// TIA Portal project "Omogenizator Miere V18" (V18)

(* hardware
DEVICE "S7-1200 station_1"  S7-1200 Station
   slot 0: "Rack_0"  S7-1200 Rack  Rack  V1.0
   slot 1: "PLC_1"  CPU 1215C DC/DC/Rly  6ES7 215-1HG40-0XB0  V4.6
DEVICE "HMI_1"  TP700 Comfort
   slot 0: "HMI_1"  TP700 Comfort  6AV2 124-0GC01-0AX0  17.0.0.0
   slot 1: "HMI_RT_1"  TP700 Comfort  6AV2 124-0GC01-0AX0  17.0.0.0
   slot 5: "HMI_1.IE_CP_1"  PROFINET Interface  17.0.0.0
      slot 1: "PROFINET Interface_1"  PROFINET Interface
         slot 1: "Port_1"  Port
         slot 2: "Port_2"  Port
   slot 7: "HMI_1.MPI/DP_CP_1"  MPI/DP Interface  17.0.0.0
DEVICE "SINAMICS G_1"  Sinamics.Device
   slot 0: "Drive_1"  G120 CU240E-2 PN-F  6SL3244-0BB13-1FA0  4.7.13
      slot 1: "PROFINET interface"  MDD-SinamicsG120-P
   slot 0: "	_0"  Rail  SinamicsG120RackPN
   slot 3: "PM240 IP20"  PM240 IP20  6SL3224-0BE25-5AA0  -
*)

// ===== PLC "PLC_1"  CPU 1215C DC/DC/Rly =====

VAR_GLOBAL   // PLC tag table "Default tag table"
   "Clock_Byte" AT %MB0 : Byte;
   "Clock_10Hz" AT %M0.0 : Bool;
   "Clock_5Hz" AT %M0.1 : Bool;
   "Clock_2.5Hz" AT %M0.2 : Bool;
   "Clock_2Hz" AT %M0.3 : Bool;
   "Clock_1.25Hz" AT %M0.4 : Bool;
   "Clock_1Hz" AT %M0.5 : Bool;
   "Clock_0.625Hz" AT %M0.6 : Bool;
   "Clock_0.5Hz" AT %M0.7 : Bool;
END_VAR

VAR_GLOBAL   // PLC tag table "Temperatura"
   "Valva incalzire" AT %Q0.1 : Bool;
END_VAR

VAR_GLOBAL   // PLC tag table "Mixer"
   "Avarie mixer" AT %I0.3 : Bool;
   "Mixer" AT %Q0.0 : Bool;
   "Viteza Mixer" AT %QW258 : Int;
   "Autorizatie_0" AT %Q257.2 : Bool;
   "Autorizatie_1" AT %Q256.1 : Bool;
   "Autorizatie_2" AT %Q256.2 : Bool;
   "Autorizatie_3" AT %Q256.3 : Bool;
   "Autorizatie_4" AT %Q256.4 : Bool;
   "Autorizatie_5" AT %Q256.5 : Bool;
   "Autorizatie_6" AT %Q256.6 : Bool;
   "Autorizatie_7" AT %Q256.7 : Bool;
   "Motor Pornit" AT %Q256.0 : Bool;
END_VAR

VAR_GLOBAL   // PLC tag table "Urgenta"
   "Buton urgenta" AT %I0.0 : Bool;
END_VAR

VAR_GLOBAL   // PLC tag table "Senzori"
   "Usa 1" AT %I0.1 : Bool;
   "Usa 2" AT %I0.2 : Bool;
   "Senzor temperatura" AT %IW64 : Int;
   "Senzor nivel" AT %IW66 : Int;
END_VAR

DATA_BLOCK "Valori Temporare"   // DB1
{ S7_Optimized_Access := 'TRUE' }
VERSION : 0.1
   VAR
      "Finalizare Program" : Bool;
      "Temporizare Setata Scursa" : Bool;
      "Alarma Usi Deschise" : Int;
      "Start/Stop" : Bool;
      "Setare Temperatura Manual" : Bool;
      "Mod Automat" : Bool;
      "Counter Temporizator Invers" : Int;
      "Setare Temporizator" : Int := 5;
      "Temperatura Setata" : Int := 35;
      "Frecventa Mixer" : Int;
      "Alarma  Senzor Temperatura" : Int;
      "Alarma Generala" : Bool;
      "Alarma Senzor Presiune" : Int;
      "Alarma Mixer" : Int;
      "Counter Nivel Presiune" : Int;
      "Usi inchise" : Bool;
      "Valoare Analog Intrare Temperatura" : Int;
      "Valoare Analog Intrare Miere" : Int;
      "Nivel Temperatura Grade" : Real;
      "Nivel Miere in Kg" : Real;
      "Buton Motor" : Bool;
      "Semafor Mixer" : Bool;
      "Pornire Mixer Manual" : Bool;
   END_VAR
BEGIN
END_DATA_BLOCK

DATA_BLOCK "Usi Inchise_DB"   // DB5
{ S7_Optimized_Access := 'TRUE' }
VERSION : 0.1
// stored: InstanceOfName Usi Inchise
"Usi Inchise"
BEGIN
   "Usa jos" := false;
   "Usa sus" := false;
END_DATA_BLOCK

// folder: System blocks/Program resources

DATA_BLOCK "IEC_Counter_Nivel_Temperatura_Crestere_DB"   // DB2
{ S7_Optimized_Access := 'TRUE' }
AUTHOR : Simatic
FAMILY : IEC
NAME : CNTR
VERSION : 1.0
// stored: InstanceOfName IEC_COUNTER
"IEC_COUNTER"
BEGIN
END_DATA_BLOCK

DATA_BLOCK "IEC_Counter_Mixer_DB"   // DB3
{ S7_Optimized_Access := 'TRUE' }
AUTHOR : Simatic
FAMILY : IEC
NAME : CNTR
VERSION : 1.0
// stored: InstanceOfName IEC_COUNTER
"IEC_COUNTER"
BEGIN
END_DATA_BLOCK

DATA_BLOCK "IEC_Counter_Temporizator_Mixer_DB"   // DB4
{ S7_Optimized_Access := 'TRUE' }
AUTHOR : Simatic
FAMILY : IEC
NAME : CNTR
VERSION : 1.0
// stored: InstanceOfName IEC_COUNTER
"IEC_COUNTER"
BEGIN
END_DATA_BLOCK

DATA_BLOCK "IEC_Counter_Nivel_Presiune_DB"   // DB6
{ S7_Optimized_Access := 'TRUE' }
AUTHOR : Simatic
FAMILY : IEC
NAME : CNTR
VERSION : 1.0
// stored: InstanceOfName IEC_COUNTER
"IEC_COUNTER"
BEGIN
END_DATA_BLOCK

// folder: (top level)

FUNCTION_BLOCK "Usi Inchise"   // FB1, LAD
{ S7_Optimized_Access := 'TRUE' }
VERSION : 0.1
   VAR_INPUT
      "Usa jos" : Bool := true;
      "Usa sus" : Bool := true;
   END_VAR
   VAR_OUTPUT
      "Usi inchise" : Bool;
   END_VAR
BEGIN

REGION Network 1: Ambele usi inchise
   // Ambii senzori returneaza true daca usile sunt inchise
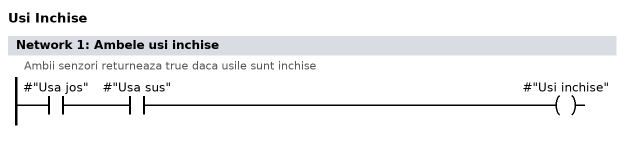
   RUNG wire#powerrail
      Contact( #"Usa jos" )
      Contact( #"Usa sus" )
      Coil( #"Usi inchise" )
   END_RUNG
   // the same network as SCL:
   #"Usi inchise" := #"Usa jos" AND #"Usa sus";
END_REGION
END_FUNCTION_BLOCK

FUNCTION "Incalzire Rezervor" : Void   // FC1, LAD
{ S7_Optimized_Access := 'TRUE' }
VERSION : 0.1
   VAR_INPUT
      "Nivel Temperatura Grade" : Int;
      "Temperatura Setata" : Int;
   END_VAR
   VAR_OUTPUT
      "Valoare Analog Intrare Temperatura" : Int;
   END_VAR
   VAR_TEMP
      "Counter Nivel Temperatura" : Int;
   END_VAR
BEGIN

REGION Network 1: Incalzire rezervor
   // Valva de incalzire este activata si se ajunge la temperatura dorita in 10 secunde(in acest caz simulat).
   // Cat timp temperatura setata nu este atinsa trimitem valori pornind de la 0 pana 27648 catre functia de procesare a valorilor analog de intrare pentru senzorul de temperatura.
   // Acest network e folosit doar pentru simulare, in realitate senzorul de temperatura trimite aceste date.
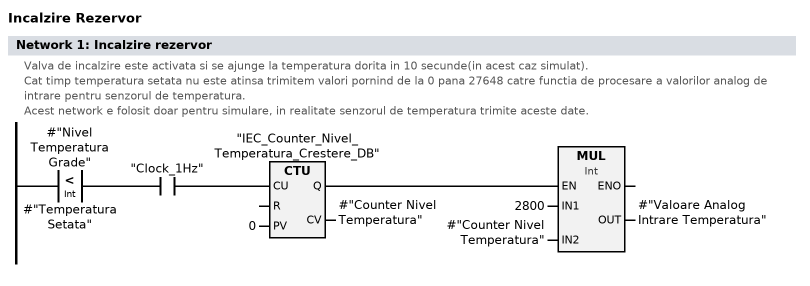
   "IEC_Counter_Nivel_Temperatura_Crestere_DB".CTU(CU := (#"Nivel Temperatura Grade" < #"Temperatura Setata") AND "Clock_1Hz",
                           PV := 0,
                           CV => #"Counter Nivel Temperatura");
   IF "IEC_Counter_Nivel_Temperatura_Crestere_DB".Q THEN
       #"Valoare Analog Intrare Temperatura" := 2800 * #"Counter Nivel Temperatura";
   END_IF;
END_REGION
END_FUNCTION

FUNCTION "Motor Exemplu" : Void   // FC2, LAD
{ S7_Optimized_Access := 'TRUE' }
VERSION : 0.1
   VAR_INPUT
      "Frecventa Mixer" : Int;
      "Buton Motor" : Bool;
   END_VAR
   VAR_OUTPUT
      "Viteza Motor" : Int;
   END_VAR
   VAR_TEMP
      "Rotatii Per Minut" : Int;
      "Valoare Procentaj Viteza" : Int;
      "Viteza Motor Exemplu" : Int;
      "Valoare Procentaj Frecventa" : Int;
   END_VAR
   VAR CONSTANT
      TempVal : Bool := true;
   END_VAR
BEGIN

REGION Network 1: Normalizarea INPUT-ului si transformarea acesteia in valoare de INPUT pentru motor(G120 DRIVE)
   // NORM_X 1500 -> Viteza de referinta amotorului(In acest caz sa zicem ca e setata din HMI)
   // SCALE_X 16348 -> Valoarea maxima care va deveni valoare INPUT pentru motor(G120 DRIVE)
   // Acest Network ar merge daca ar exista un motor/drive fizic. Aici e folosit strict ca exemplu.
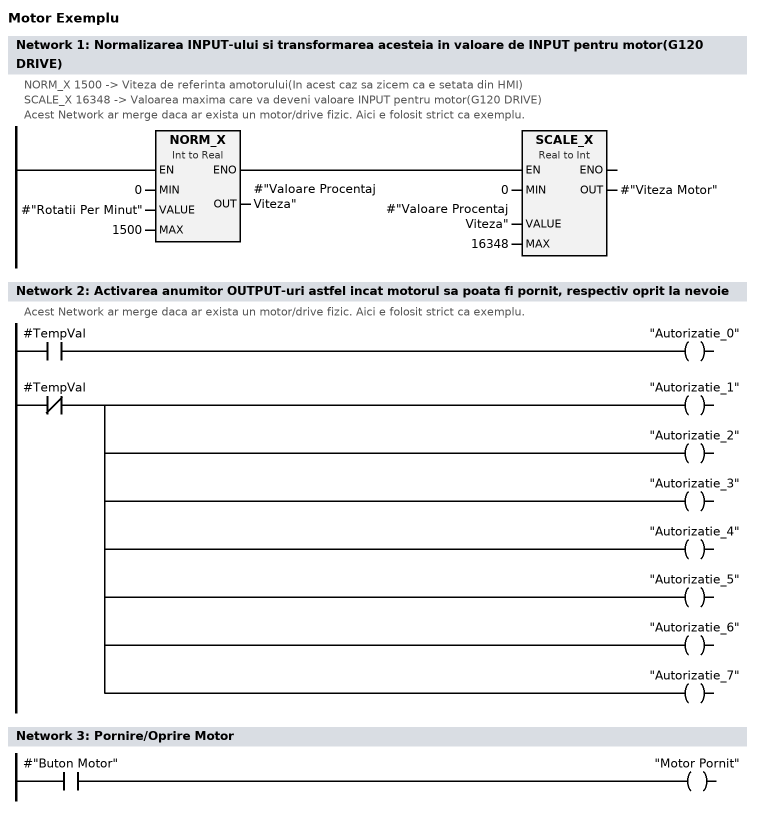
   RUNG wire#powerrail
      { S7_Templates := "[SrcType := Int, DestType := Real]" } Normalize(min := 0, value := #"Rotatii Per Minut", max := 1500, out => #"Valoare Procentaj Viteza")
      { S7_Templates := "[SrcType := Real, DestType := Int]" } Scale(min := 0, value := #"Valoare Procentaj Viteza", max := 16348, out => #"Viteza Motor")
   END_RUNG
   // the same network as SCL:
   #"Valoare Procentaj Viteza" := NORM_X(MIN := 0, VALUE := #"Rotatii Per Minut", MAX := 1500);
   #"Viteza Motor" := SCALE_X(MIN := 0, VALUE := #"Valoare Procentaj Viteza", MAX := 16348);
END_REGION

REGION Network 2: Activarea anumitor OUTPUT-uri astfel incat motorul sa poata fi pornit, respectiv oprit la nevoie
   // Acest Network ar merge daca ar exista un motor/drive fizic. Aici e folosit strict ca exemplu.
   RUNG wire#powerrail
      Contact( #TempVal )
      Coil( "Autorizatie_0" )
   END_RUNG
   RUNG wire#powerrail
      I_Contact( #TempVal )
      wire#w1
      Coil( "Autorizatie_1" )
   END_RUNG
   RUNG wire#w1
      Coil( "Autorizatie_2" )
   END_RUNG
   RUNG wire#w1
      Coil( "Autorizatie_3" )
   END_RUNG
   RUNG wire#w1
      Coil( "Autorizatie_4" )
   END_RUNG
   RUNG wire#w1
      Coil( "Autorizatie_5" )
   END_RUNG
   RUNG wire#w1
      Coil( "Autorizatie_6" )
   END_RUNG
   RUNG wire#w1
      Coil( "Autorizatie_7" )
   END_RUNG
   // the same network as SCL:
   "Autorizatie_0" := #TempVal;
   "Autorizatie_1" := NOT #TempVal;
   "Autorizatie_2" := NOT #TempVal;
   "Autorizatie_3" := NOT #TempVal;
   "Autorizatie_4" := NOT #TempVal;
   "Autorizatie_5" := NOT #TempVal;
   "Autorizatie_6" := NOT #TempVal;
   "Autorizatie_7" := NOT #TempVal;
END_REGION

REGION Network 3: Pornire/Oprire Motor
   RUNG wire#powerrail
      Contact( #"Buton Motor" )
      Coil( "Motor Pornit" )
   END_RUNG
   // the same network as SCL:
   "Motor Pornit" := #"Buton Motor";
END_REGION
END_FUNCTION

FUNCTION "Motor_Proxy" : Void   // FC3, LAD
{ S7_Optimized_Access := 'TRUE' }
VERSION : 0.1
   VAR_OUTPUT
      "Frecventa Motor" : Int;   // 50 Hz(1500RotatiiPerMinut) conform setarilor facute in Device-ul Drive G120
   END_VAR
   VAR_TEMP
      "Counter Mixer" : Int;
      Frecventa : Int;
      "Semafor counter" : Bool;
   END_VAR
BEGIN

REGION Network 1: Pornirea Mixerului
   // Mixerul porneste si ajunge in timpul de 10 secunde(timp setat in acest caz simulat) la viteza de 50Hz(1500 rotatii per minut)
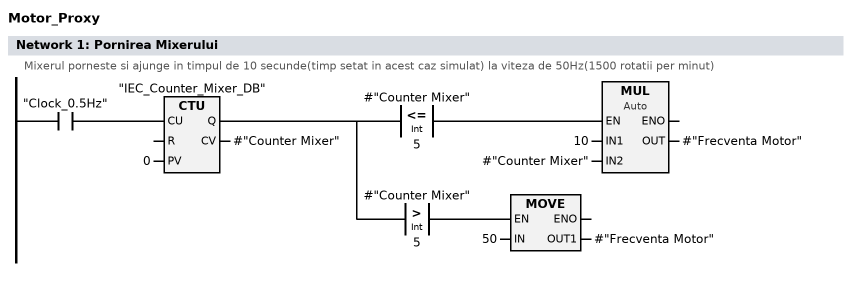
   "IEC_Counter_Mixer_DB".CTU(CU := "Clock_0.5Hz", PV := 0, CV => #"Counter Mixer");
   IF "IEC_Counter_Mixer_DB".Q AND (#"Counter Mixer" <= 5) THEN
       #"Frecventa Motor" := 10 * #"Counter Mixer";
   END_IF;
   IF "IEC_Counter_Mixer_DB".Q AND (#"Counter Mixer" > 5) THEN #"Frecventa Motor" := 50; END_IF;
END_REGION
END_FUNCTION

FUNCTION "Procesare Intrari Analog Senzor Miere" : Void   // FC4, LAD
{ S7_Optimized_Access := 'TRUE' }
VERSION : 0.1
   VAR_INPUT
      "Valoare Intrare Analog" : Int;
   END_VAR
   VAR_OUTPUT
      "Valoare Nivel Miere in KG" : Real;
   END_VAR
   VAR_TEMP
      "Nivel Miere Procentaj" : Real;
   END_VAR
   VAR CONSTANT
      "Valoare Maxima Intrare Analog" : Int := 27648;
      "Cantitatea de Miere Introdusa" : Real := 11157.0;
   END_VAR
BEGIN

REGION Network 1: Normalizarea Valorii Analog de Intrare
   // Valorile Analog de intrare la PLC sunt intre 0 si 27648(Int)
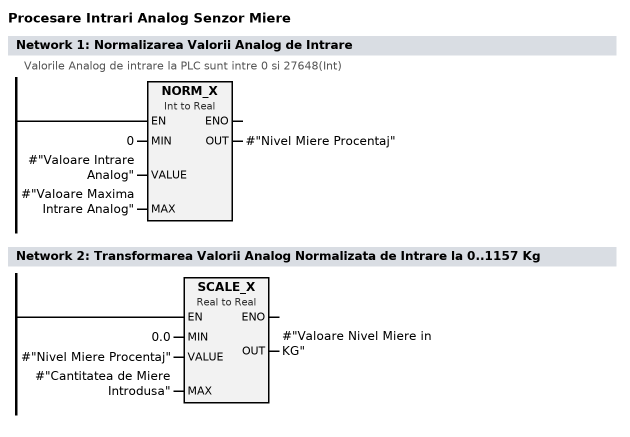
   RUNG wire#powerrail
      { S7_Templates := "[SrcType := Int, DestType := Real]" } Normalize(min := 0, value := #"Valoare Intrare Analog", max := #"Valoare Maxima Intrare Analog", out => #"Nivel Miere Procentaj")
   END_RUNG
   // the same network as SCL:
   #"Nivel Miere Procentaj" := NORM_X(MIN := 0, VALUE := #"Valoare Intrare Analog", MAX := #"Valoare Maxima Intrare Analog");
END_REGION

REGION Network 2: Transformarea Valorii Analog Normalizata de Intrare la 0..1157 Kg
   RUNG wire#powerrail
      { S7_Templates := "[SrcType := Real, DestType := Real]" } Scale(min := 0.0, value := #"Nivel Miere Procentaj", max := #"Cantitatea de Miere Introdusa", out => #"Valoare Nivel Miere in KG")
   END_RUNG
   // the same network as SCL:
   #"Valoare Nivel Miere in KG" := SCALE_X(MIN := 0.0, VALUE := #"Nivel Miere Procentaj", MAX := #"Cantitatea de Miere Introdusa");
END_REGION
END_FUNCTION

FUNCTION "Procesare Intrari Analog Senzor Temperatura" : Void   // FC5, LAD
{ S7_Optimized_Access := 'TRUE' }
VERSION : 0.1
   VAR_INPUT
      "Temperatura Setata" : Int;
      "Valoare Intrare Analog" : Int;
   END_VAR
   VAR_OUTPUT
      "Nivel Temperatura in Grade" : Real;
   END_VAR
   VAR_TEMP
      "Temp Setata" : Real;
      "Nivel Temperatura Procentaj" : Real;
   END_VAR
   VAR CONSTANT
      "Valoare Maxima Intrare Analog" : Int := 27648;
   END_VAR
BEGIN

REGION Network 1: Normalizarea Valorii Analog de Intrare
   // Valorile Analog de intrare la PLC sunt intre 0 si 27648(Int)
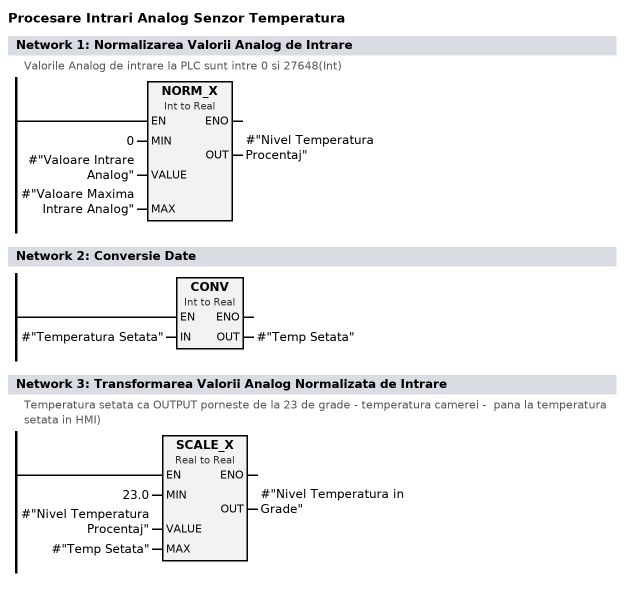
   RUNG wire#powerrail
      { S7_Templates := "[SrcType := Int, DestType := Real]" } Normalize(min := 0, value := #"Valoare Intrare Analog", max := #"Valoare Maxima Intrare Analog", out => #"Nivel Temperatura Procentaj")
   END_RUNG
   // the same network as SCL:
   #"Nivel Temperatura Procentaj" := NORM_X(MIN := 0, VALUE := #"Valoare Intrare Analog", MAX := #"Valoare Maxima Intrare Analog");
END_REGION

REGION Network 2: Conversie Date
   RUNG wire#powerrail
      { S7_Templates := "[SrcType := Int, DestType := Real]" } Convert(in := #"Temperatura Setata", out => #"Temp Setata")
   END_RUNG
   // the same network as SCL:
   #"Temp Setata" := INT_TO_REAL(#"Temperatura Setata");
END_REGION

REGION Network 3: Transformarea Valorii Analog Normalizata de Intrare
   // Temperatura setata ca OUTPUT porneste de la 23 de grade - temperatura camerei -  pana la temperatura setata in HMI)
   RUNG wire#powerrail
      { S7_Templates := "[SrcType := Real, DestType := Real]" } Scale(min := 23.0, value := #"Nivel Temperatura Procentaj", max := #"Temp Setata", out => #"Nivel Temperatura in Grade")
   END_RUNG
   // the same network as SCL:
   #"Nivel Temperatura in Grade" := SCALE_X(MIN := 23.0, VALUE := #"Nivel Temperatura Procentaj", MAX := #"Temp Setata");
END_REGION
END_FUNCTION

FUNCTION "Temporizator Mixer" : Void   // FC6, LAD
{ S7_Optimized_Access := 'TRUE' }
VERSION : 0.1
   VAR_INPUT
      "Temporizator Setat" : Int;
   END_VAR
   VAR_OUTPUT
      "Temporizator Invers" : Int;
   END_VAR
   VAR_TEMP
      "Variabila Temporara" : Int;
      "Counter Temporizator" : Int;
   END_VAR
BEGIN

REGION Network 1: Simulare Temporizator Mixer
   // Simulare in care scadem din timpul setat, cu 1 la fiecare secunda pana ajungem la 0 ca apoi sa putem afisa finalitatea procesului de omogenizare.
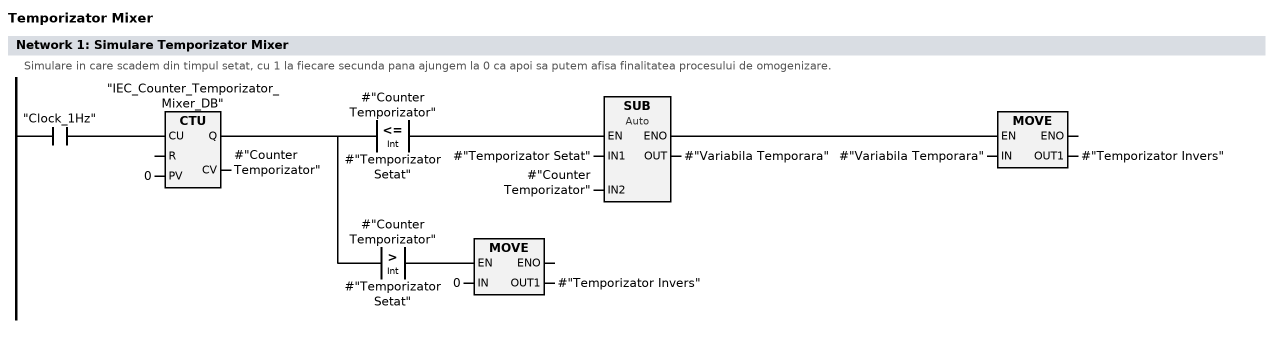
   "IEC_Counter_Temporizator_Mixer_DB".CTU(CU := "Clock_1Hz", PV := 0, CV => #"Counter Temporizator");
   IF "IEC_Counter_Temporizator_Mixer_DB".Q AND (#"Counter Temporizator" <= #"Temporizator Setat") THEN
       #"Variabila Temporara" := #"Temporizator Setat" - #"Counter Temporizator";
       #"Temporizator Invers" := #"Variabila Temporara";
   END_IF;
   IF "IEC_Counter_Temporizator_Mixer_DB".Q AND (#"Counter Temporizator" > #"Temporizator Setat") THEN
       #"Temporizator Invers" := 0;
   END_IF;
END_REGION
END_FUNCTION

ORGANIZATION_BLOCK "Main"   // OB1, LAD, ProgramCycle
TITLE = "Main Program Sweep (Cycle)"
{ S7_Optimized_Access := 'TRUE' }
VERSION : 0.1
   VAR_INPUT
      Initial_Call : Bool;   // Initial call of this OB
      Remanence : Bool;   // =True, if remanent data are available
   END_VAR
   VAR CONSTANT
      "Inserare Miere 5 Secunde" : Int := 5530;
   END_VAR
   VAR_TEMP   // added for the SCL form of the ladder/FBD networks
      _w1 : Bool;
   END_VAR
BEGIN

REGION Network 1: Procesare Intrari Analog Senzor Miere
   // In PLC ar trebui sa intre in INPUT date de la senzorul de presiune(nivel) al rezervorului ca apoi sa procesam datele si sa aratam in HMI(ecran) nivelul rezervorului in Kg.
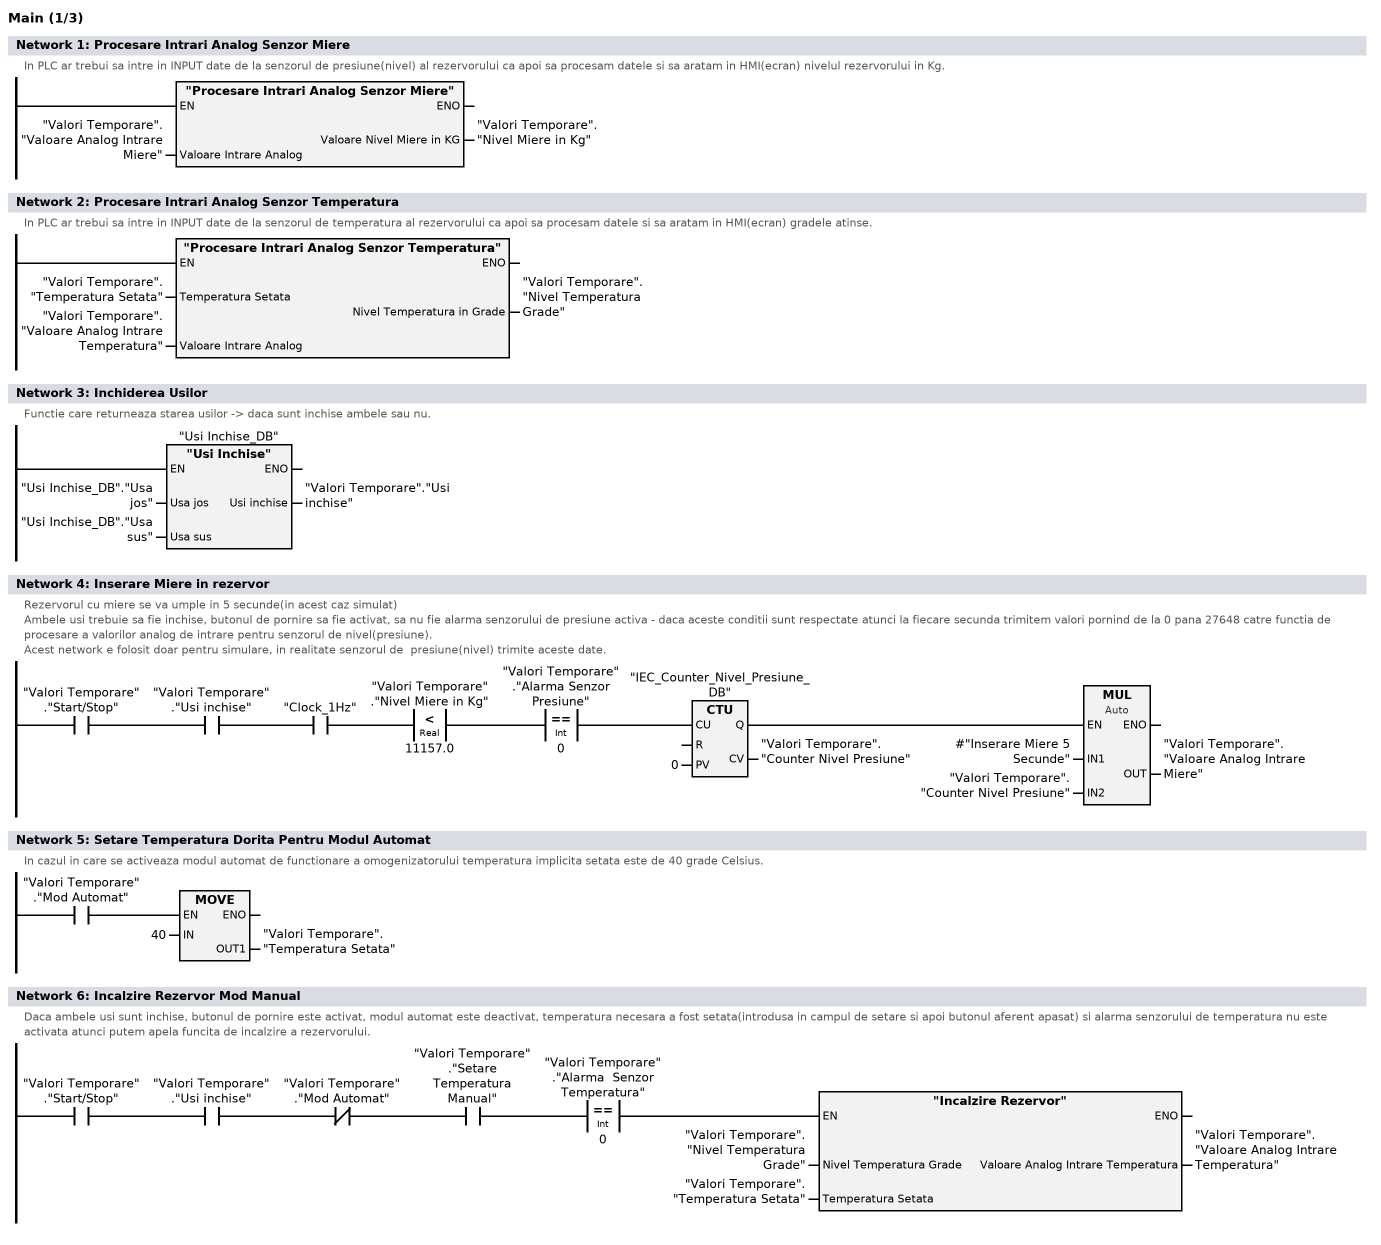
   RUNG wire#powerrail
      "Procesare Intrari Analog Senzor Miere"("Valoare Intrare Analog" := "Valori Temporare"."Valoare Analog Intrare Miere", "Valoare Nivel Miere in KG" => "Valori Temporare"."Nivel Miere in Kg")
   END_RUNG
   // the same network as SCL:
   "Procesare Intrari Analog Senzor Miere"("Valoare Intrare Analog" := "Valori Temporare"."Valoare Analog Intrare Miere",
                           "Valoare Nivel Miere in KG" => "Valori Temporare"."Nivel Miere in Kg");
END_REGION

REGION Network 2: Procesare Intrari Analog Senzor Temperatura
   // In PLC ar trebui sa intre in INPUT date de la senzorul de temperatura al rezervorului ca apoi sa procesam datele si sa aratam in HMI(ecran) gradele atinse.
   RUNG wire#powerrail
      "Procesare Intrari Analog Senzor Temperatura"("Temperatura Setata" := "Valori Temporare"."Temperatura Setata", "Valoare Intrare Analog" := "Valori Temporare"."Valoare Analog Intrare Temperatura", "Nivel Temperatura in Grade" => "Valori Temporare"."Nivel Temperatura Grade")
   END_RUNG
   // the same network as SCL:
   "Procesare Intrari Analog Senzor Temperatura"("Temperatura Setata" := "Valori Temporare"."Temperatura Setata",
                           "Valoare Intrare Analog" := "Valori Temporare"."Valoare Analog Intrare Temperatura",
                           "Nivel Temperatura in Grade" => "Valori Temporare"."Nivel Temperatura Grade");
END_REGION

REGION Network 3: Inchiderea Usilor
   // Functie care returneaza starea usilor -> daca sunt inchise ambele sau nu.
   RUNG wire#powerrail
      "Usi Inchise_DB"("Usa jos" := "Usi Inchise_DB"."Usa jos", "Usa sus" := "Usi Inchise_DB"."Usa sus", "Usi inchise" => "Valori Temporare"."Usi inchise")
   END_RUNG
   // the same network as SCL:
   "Usi Inchise_DB"("Usa jos" := "Usi Inchise_DB"."Usa jos",   // "Usi Inchise"
                    "Usa sus" := "Usi Inchise_DB"."Usa sus",
                    "Usi inchise" => "Valori Temporare"."Usi inchise");
END_REGION

REGION Network 4: Inserare Miere in rezervor
   // Rezervorul cu miere se va umple in 5 secunde(in acest caz simulat)
   // Ambele usi trebuie sa fie inchise, butonul de pornire sa fie activat, sa nu fie alarma senzorului de presiune activa - daca aceste conditii sunt respectate atunci la fiecare secunda trimitem valori pornind de la 0 pana 27648 catre functia de procesare a valorilor analog de intrare pentru senzorul de nivel(presiune).
   // Acest network e folosit doar pentru simulare, in realitate senzorul de  presiune(nivel) trimite aceste date.
   "IEC_Counter_Nivel_Presiune_DB".CTU(CU := "Valori Temporare"."Start/Stop" AND "Valori Temporare"."Usi inchise" AND "Clock_1Hz" AND ("Valori Temporare"."Nivel Miere in Kg" < 11157.0) AND ("Valori Temporare"."Alarma Senzor Presiune" = 0),
                           PV := 0,
                           CV => "Valori Temporare"."Counter Nivel Presiune");
   IF "IEC_Counter_Nivel_Presiune_DB".Q THEN
       "Valori Temporare"."Valoare Analog Intrare Miere" := #"Inserare Miere 5 Secunde" * "Valori Temporare"."Counter Nivel Presiune";
   END_IF;
END_REGION

REGION Network 5: Setare Temperatura Dorita Pentru Modul Automat
   // In cazul in care se activeaza modul automat de functionare a omogenizatorului temperatura implicita setata este de 40 grade Celsius.
   RUNG wire#powerrail
      Contact( "Valori Temporare"."Mod Automat" )
      Move(in := 40, out1 => "Valori Temporare"."Temperatura Setata")
   END_RUNG
   // the same network as SCL:
   IF "Valori Temporare"."Mod Automat" THEN "Valori Temporare"."Temperatura Setata" := 40; END_IF;
END_REGION

REGION Network 6: Incalzire Rezervor Mod Manual
   // Daca ambele usi sunt inchise, butonul de pornire este activat, modul automat este deactivat, temperatura necesara a fost setata(introdusa in campul de setare si apoi butonul aferent apasat) si alarma senzorului de temperatura nu este activata atunci putem apela funcita de incalzire a rezervorului.
   RUNG wire#powerrail
      Contact( "Valori Temporare"."Start/Stop" )
      Contact( "Valori Temporare"."Usi inchise" )
      I_Contact( "Valori Temporare"."Mod Automat" )
      Contact( "Valori Temporare"."Setare Temperatura Manual" )
      { S7_Templates := "SrcType := Int" } EQ_Contact(in1 := "Valori Temporare"."Alarma  Senzor Temperatura", in2 := 0)
      "Incalzire Rezervor"("Nivel Temperatura Grade" := "Valori Temporare"."Nivel Temperatura Grade", "Temperatura Setata" := "Valori Temporare"."Temperatura Setata", "Valoare Analog Intrare Temperatura" => "Valori Temporare"."Valoare Analog Intrare Temperatura")
   END_RUNG
   // the same network as SCL:
   IF "Valori Temporare"."Start/Stop" AND "Valori Temporare"."Usi inchise" AND NOT "Valori Temporare"."Mod Automat" AND "Valori Temporare"."Setare Temperatura Manual" AND ("Valori Temporare"."Alarma  Senzor Temperatura" = 0) THEN
       "Incalzire Rezervor"("Nivel Temperatura Grade" := "Valori Temporare"."Nivel Temperatura Grade",
                            "Temperatura Setata" := "Valori Temporare"."Temperatura Setata",
                            "Valoare Analog Intrare Temperatura" => "Valori Temporare"."Valoare Analog Intrare Temperatura");
   END_IF;
END_REGION

REGION Network 7: Incalzire Rezervor Mod Automat
   // Daca ambele usi sunt inchise, butonul de pornire este activat, modul automat este activat si alarma senzorului de temperatura nu este activata atunci putem apela funcita de incalzire a rezervorului.
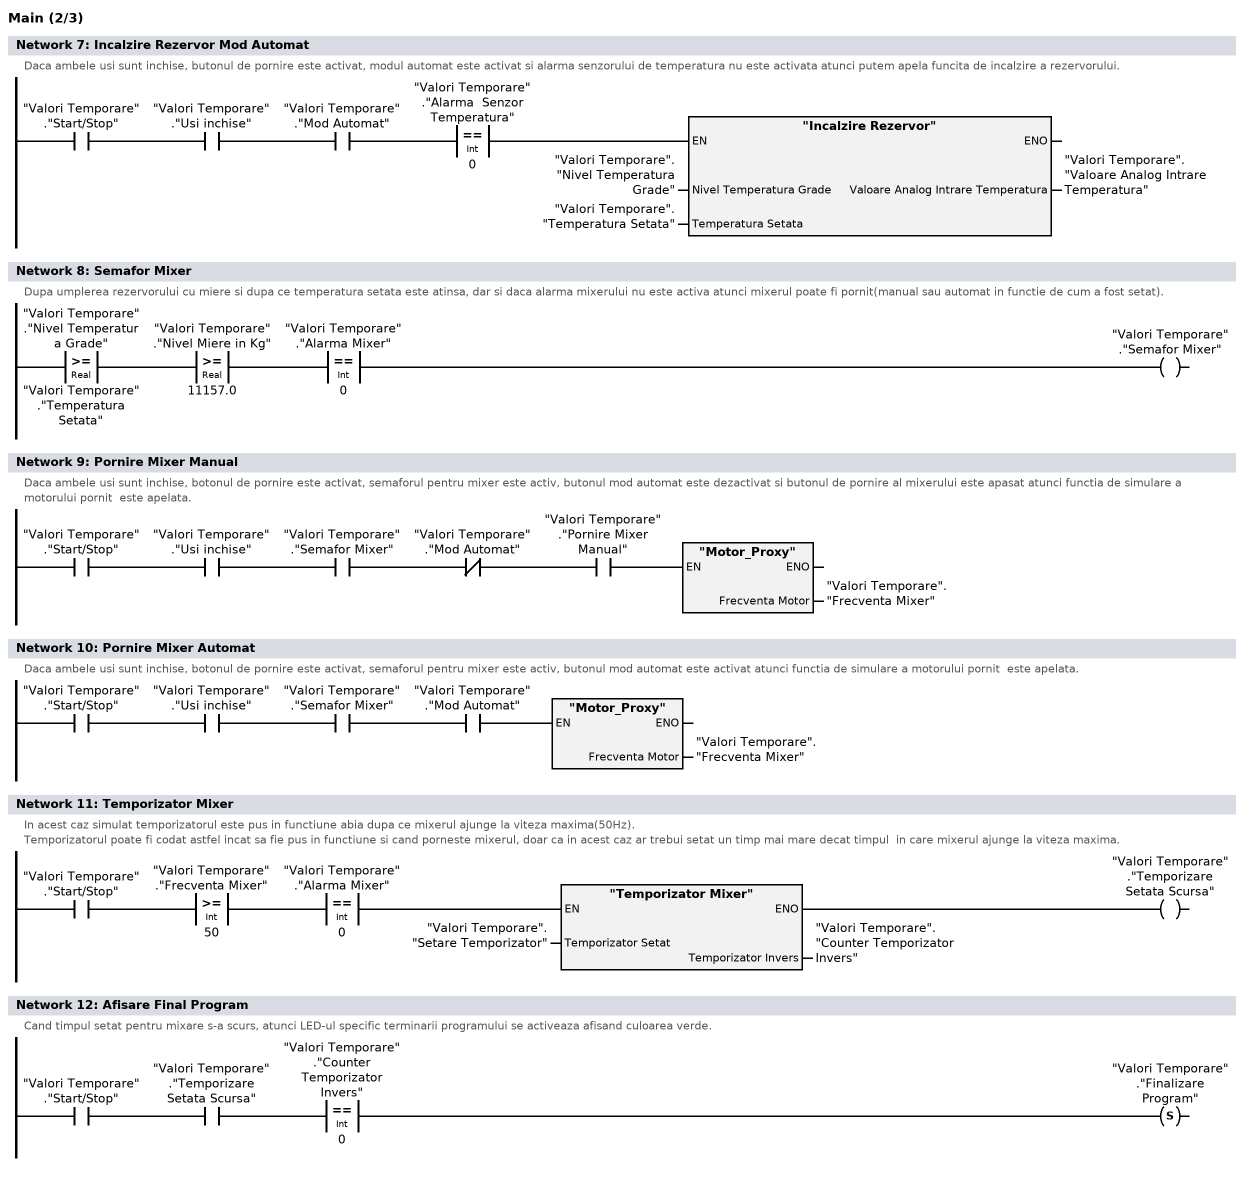
   RUNG wire#powerrail
      Contact( "Valori Temporare"."Start/Stop" )
      Contact( "Valori Temporare"."Usi inchise" )
      Contact( "Valori Temporare"."Mod Automat" )
      { S7_Templates := "SrcType := Int" } EQ_Contact(in1 := "Valori Temporare"."Alarma  Senzor Temperatura", in2 := 0)
      "Incalzire Rezervor"("Nivel Temperatura Grade" := "Valori Temporare"."Nivel Temperatura Grade", "Temperatura Setata" := "Valori Temporare"."Temperatura Setata", "Valoare Analog Intrare Temperatura" => "Valori Temporare"."Valoare Analog Intrare Temperatura")
   END_RUNG
   // the same network as SCL:
   IF "Valori Temporare"."Start/Stop" AND "Valori Temporare"."Usi inchise" AND "Valori Temporare"."Mod Automat" AND ("Valori Temporare"."Alarma  Senzor Temperatura" = 0) THEN
       "Incalzire Rezervor"("Nivel Temperatura Grade" := "Valori Temporare"."Nivel Temperatura Grade",
                            "Temperatura Setata" := "Valori Temporare"."Temperatura Setata",
                            "Valoare Analog Intrare Temperatura" => "Valori Temporare"."Valoare Analog Intrare Temperatura");
   END_IF;
END_REGION

REGION Network 8: Semafor Mixer
   // Dupa umplerea rezervorului cu miere si dupa ce temperatura setata este atinsa, dar si daca alarma mixerului nu este activa atunci mixerul poate fi pornit(manual sau automat in functie de cum a fost setat).
   RUNG wire#powerrail
      { S7_Templates := "SrcType := Real" } GE_Contact(in1 := "Valori Temporare"."Nivel Temperatura Grade", in2 := "Valori Temporare"."Temperatura Setata")
      { S7_Templates := "SrcType := Real" } GE_Contact(in1 := "Valori Temporare"."Nivel Miere in Kg", in2 := 11157.0)
      { S7_Templates := "SrcType := Int" } EQ_Contact(in1 := "Valori Temporare"."Alarma Mixer", in2 := 0)
      Coil( "Valori Temporare"."Semafor Mixer" )
   END_RUNG
   // the same network as SCL:
   "Valori Temporare"."Semafor Mixer" := ("Valori Temporare"."Nivel Temperatura Grade" >= "Valori Temporare"."Temperatura Setata") AND ("Valori Temporare"."Nivel Miere in Kg" >= 11157.0) AND ("Valori Temporare"."Alarma Mixer" = 0);
END_REGION

REGION Network 9: Pornire Mixer Manual
   // Daca ambele usi sunt inchise, botonul de pornire este activat, semaforul pentru mixer este activ, butonul mod automat este dezactivat si butonul de pornire al mixerului este apasat atunci functia de simulare a motorului pornit  este apelata.
   RUNG wire#powerrail
      Contact( "Valori Temporare"."Start/Stop" )
      Contact( "Valori Temporare"."Usi inchise" )
      Contact( "Valori Temporare"."Semafor Mixer" )
      I_Contact( "Valori Temporare"."Mod Automat" )
      Contact( "Valori Temporare"."Pornire Mixer Manual" )
      "Motor_Proxy"("Frecventa Motor" => "Valori Temporare"."Frecventa Mixer")
   END_RUNG
   // the same network as SCL:
   IF "Valori Temporare"."Start/Stop" AND "Valori Temporare"."Usi inchise" AND "Valori Temporare"."Semafor Mixer" AND NOT "Valori Temporare"."Mod Automat" AND "Valori Temporare"."Pornire Mixer Manual" THEN
       "Motor_Proxy"("Frecventa Motor" => "Valori Temporare"."Frecventa Mixer");
   END_IF;
END_REGION

REGION Network 10: Pornire Mixer Automat
   // Daca ambele usi sunt inchise, botonul de pornire este activat, semaforul pentru mixer este activ, butonul mod automat este activat atunci functia de simulare a motorului pornit  este apelata.
   RUNG wire#powerrail
      Contact( "Valori Temporare"."Start/Stop" )
      Contact( "Valori Temporare"."Usi inchise" )
      Contact( "Valori Temporare"."Semafor Mixer" )
      Contact( "Valori Temporare"."Mod Automat" )
      "Motor_Proxy"("Frecventa Motor" => "Valori Temporare"."Frecventa Mixer")
   END_RUNG
   // the same network as SCL:
   IF "Valori Temporare"."Start/Stop" AND "Valori Temporare"."Usi inchise" AND "Valori Temporare"."Semafor Mixer" AND "Valori Temporare"."Mod Automat" THEN
       "Motor_Proxy"("Frecventa Motor" => "Valori Temporare"."Frecventa Mixer");
   END_IF;
END_REGION

REGION Network 11: Temporizator Mixer
   // In acest caz simulat temporizatorul este pus in functiune abia dupa ce mixerul ajunge la viteza maxima(50Hz).
   // Temporizatorul poate fi codat astfel incat sa fie pus in functiune si cand porneste mixerul, doar ca in acest caz ar trebui setat un timp mai mare decat timpul  in care mixerul ajunge la viteza maxima.
   RUNG wire#powerrail
      Contact( "Valori Temporare"."Start/Stop" )
      { S7_Templates := "SrcType := Int" } GE_Contact(in1 := "Valori Temporare"."Frecventa Mixer", in2 := 50)
      { S7_Templates := "SrcType := Int" } EQ_Contact(in1 := "Valori Temporare"."Alarma Mixer", in2 := 0)
      "Temporizator Mixer"("Temporizator Setat" := "Valori Temporare"."Setare Temporizator", "Temporizator Invers" => "Valori Temporare"."Counter Temporizator Invers")
      Coil( "Valori Temporare"."Temporizare Setata Scursa" )
   END_RUNG
   // the same network as SCL:
   "Temporizator Mixer"(EN := "Valori Temporare"."Start/Stop" AND ("Valori Temporare"."Frecventa Mixer" >= 50) AND ("Valori Temporare"."Alarma Mixer" = 0),
                        "Temporizator Setat" := "Valori Temporare"."Setare Temporizator",
                        "Temporizator Invers" => "Valori Temporare"."Counter Temporizator Invers",
                        ENO => #_w1);
   "Valori Temporare"."Temporizare Setata Scursa" := #_w1;
END_REGION

REGION Network 12: Afisare Final Program
   // Cand timpul setat pentru mixare s-a scurs, atunci LED-ul specific terminarii programului se activeaza afisand culoarea verde.
   RUNG wire#powerrail
      Contact( "Valori Temporare"."Start/Stop" )
      Contact( "Valori Temporare"."Temporizare Setata Scursa" )
      { S7_Templates := "SrcType := Int" } EQ_Contact(in1 := "Valori Temporare"."Counter Temporizator Invers", in2 := 0)
      S_Coil( "Valori Temporare"."Finalizare Program" )
   END_RUNG
   // the same network as SCL:
   IF "Valori Temporare"."Start/Stop" AND "Valori Temporare"."Temporizare Setata Scursa" AND ("Valori Temporare"."Counter Temporizator Invers" = 0) THEN
       "Valori Temporare"."Finalizare Program" := TRUE;
   END_IF;
END_REGION

REGION Network 13: Simulare Alarma Usi Deschise
   // Daca butonul de pornire este activat si una din usi sau ambele usi sunt deschise atunci activam alarma de usi deschise, in caz contrar dezactivam alarma.
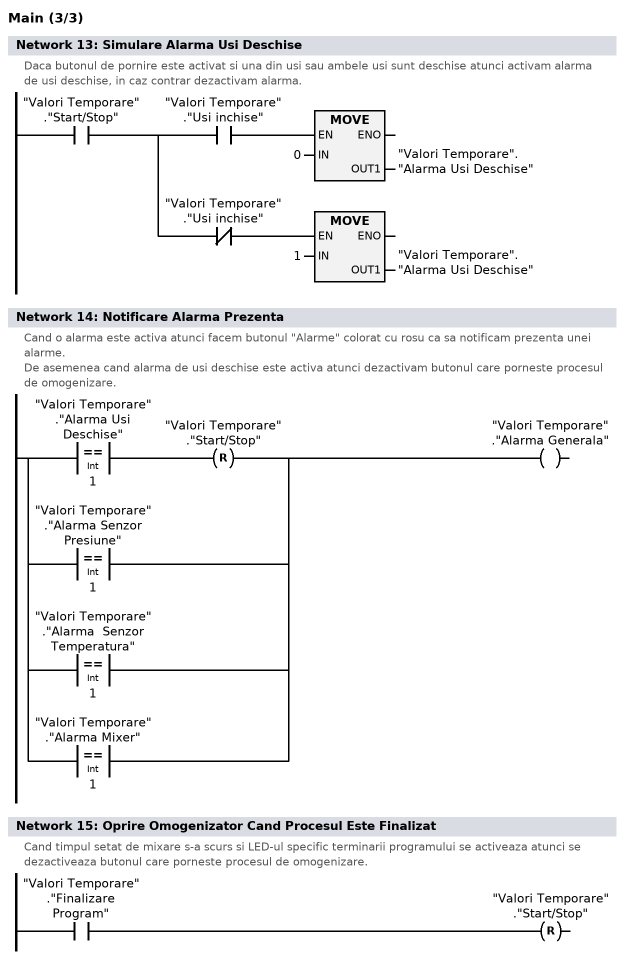
   RUNG wire#powerrail
      Contact( "Valori Temporare"."Start/Stop" )
      wire#w1
      Contact( "Valori Temporare"."Usi inchise" )
      Move(in := 0, out1 => "Valori Temporare"."Alarma Usi Deschise")
   END_RUNG
   RUNG wire#w1
      I_Contact( "Valori Temporare"."Usi inchise" )
      Move(in := 1, out1 => "Valori Temporare"."Alarma Usi Deschise")
   END_RUNG
   // the same network as SCL:
   IF "Valori Temporare"."Start/Stop" AND "Valori Temporare"."Usi inchise" THEN
       "Valori Temporare"."Alarma Usi Deschise" := 0;
   END_IF;
   IF "Valori Temporare"."Start/Stop" AND NOT "Valori Temporare"."Usi inchise" THEN
       "Valori Temporare"."Alarma Usi Deschise" := 1;
   END_IF;
END_REGION

REGION Network 14: Notificare Alarma Prezenta
   // Cand o alarma este activa atunci facem butonul "Alarme" colorat cu rosu ca sa notificam prezenta unei alarme. 
   // De asemenea cand alarma de usi deschise este activa atunci dezactivam butonul care porneste procesul de omogenizare.
   RUNG wire#powerrail
      { S7_Templates := "SrcType := Int" } EQ_Contact(in1 := "Valori Temporare"."Alarma Usi Deschise", in2 := 1)
      R_Coil( "Valori Temporare"."Start/Stop" )
      wire#w1
      Coil( "Valori Temporare"."Alarma Generala" )
   END_RUNG
   RUNG wire#powerrail
      { S7_Templates := "SrcType := Int" } EQ_Contact(in1 := "Valori Temporare"."Alarma Senzor Presiune", in2 := 1)
   END_RUNG wire#w1
   RUNG wire#powerrail
      { S7_Templates := "SrcType := Int" } EQ_Contact(in1 := "Valori Temporare"."Alarma  Senzor Temperatura", in2 := 1)
   END_RUNG wire#w1
   RUNG wire#powerrail
      { S7_Templates := "SrcType := Int" } EQ_Contact(in1 := "Valori Temporare"."Alarma Mixer", in2 := 1)
   END_RUNG wire#w1
   // the same network as SCL:
   #_w1 := "Valori Temporare"."Alarma Usi Deschise" = 1;
   IF #_w1 THEN "Valori Temporare"."Start/Stop" := FALSE; END_IF;
   "Valori Temporare"."Alarma Generala" := #_w1 OR ("Valori Temporare"."Alarma Senzor Presiune" = 1) OR ("Valori Temporare"."Alarma  Senzor Temperatura" = 1) OR ("Valori Temporare"."Alarma Mixer" = 1);
END_REGION

REGION Network 15: Oprire Omogenizator Cand Procesul Este Finalizat
   // Cand timpul setat de mixare s-a scurs si LED-ul specific terminarii programului se activeaza atunci se dezactiveaza butonul care porneste procesul de omogenizare.
   RUNG wire#powerrail
      Contact( "Valori Temporare"."Finalizare Program" )
      R_Coil( "Valori Temporare"."Start/Stop" )
   END_RUNG
   // the same network as SCL:
   IF "Valori Temporare"."Finalizare Program" THEN "Valori Temporare"."Start/Stop" := FALSE; END_IF;
END_REGION
END_ORGANIZATION_BLOCK

(* ===== HMI "HMI_RT_1" =====
system functions are stored by id; their names below are inferred from use
connection "HMI_Connection_1": ETHERNET, S7_1200_OMS

HMI tags "Default tag table"
   "Tag_ScreenNumber" : UInt, internal
   "Valori Temporare_Temperatura Setata" : Int = PLC "Valori Temporare"."Temperatura Setata", 1 s
   "Valori Temporare_Nivel Temperatura Grade" : Real = PLC "Valori Temporare"."Nivel Temperatura Grade", 1 s
   "Valori Temporare_Setare Temperatura Manual" : Bool = PLC "Valori Temporare"."Setare Temperatura Manual", 1 s
   "Valori Temporare_Mod Automat" : Bool = PLC "Valori Temporare"."Mod Automat", 1 s
   "Valori Temporare_Frecventa Mixer" : Int = PLC "Valori Temporare"."Frecventa Mixer", 1 s
   "Valori Temporare_Pornire Mixer Manual" : Bool = PLC "Valori Temporare"."Pornire Mixer Manual", 1 s
   "Valori Temporare_Setare Temporizator" : Int = PLC "Valori Temporare"."Setare Temporizator", 1 s
   "Valori Temporare_Counter Temporizator Invers" : Int = PLC "Valori Temporare"."Counter Temporizator Invers", 1 s
   "Valori Temporare_Finalizare Program" : Bool = PLC "Valori Temporare"."Finalizare Program", 1 s
   "Valori Temporare_Nivel Miere in Kg" : Real = PLC "Valori Temporare"."Nivel Miere in Kg", 1 s
   "Usi Inchise_DB_Usa jos" : Bool = PLC "Usi Inchise_DB"."Usa jos", 1 s
   "Usi Inchise_DB_Usa sus" : Bool = PLC "Usi Inchise_DB"."Usa sus", 1 s
   "Valori Temporare_Start/Stop" : Bool = PLC "Valori Temporare".Start/Stop, 1 s
   "Valori Temporare_Alarma Usi Deschise" : Int = PLC "Valori Temporare"."Alarma Usi Deschise", 1 s
   "Valori Temporare_Alarma Mixer" : Int = PLC "Valori Temporare"."Alarma Mixer", 1 s
   "Valori Temporare_Alarma Senzor Presiune" : Int = PLC "Valori Temporare"."Alarma Senzor Presiune", 1 s
   "Valori Temporare_Alarma  Senzor Temperatura" : Int = PLC "Valori Temporare"."Alarma  Senzor Temperatura", 1 s

discrete alarms
   2: 'Mixer defect! Reparatii necesare!', class Errors, trigger "Valori Temporare_Alarma Mixer" bit 0
   3: 'Senzor presiune defect! Reparatii necesare!', class Errors, trigger "Valori Temporare_Alarma Senzor Presiune" bit 0
   1: 'O usa sau ambele usi sunt deschise', class Warnings, trigger "Valori Temporare_Alarma Usi Deschise" bit 0
   4: 'Senzor temperatura defect! Reparatii necesare!', class Errors, trigger "Valori Temporare_Alarma  Senzor Temperatura" bit 0

screen "Meniu" 800x480, template "Template_1"
   on GenerateScreen: SetTag("Tag_ScreenNumber", 1)
   TextField "Text field_1" at 159,16 size 123x23; Text 'Temperatura'
   TextField "Text field_2" at 14,58 size 42x23; Text 'Set:'
   IOField "I/O field_1" at 63,56 size 96x32; FormatPattern s99999
      ProcessValue <- "Valori Temporare_Temperatura Setata"
   IOField "I/O field_2" at 179,56 size 96x32; FormatPattern s999999999.999
      ProcessValue <- "Valori Temporare_Nivel Temperatura Grade"
   TextField "Text field_3" at 286,61 size 121x23; Text 'Grade atinse'
   Bar "Bar_1" at 433,56 size 80x230; MinimumValue 0; MaximumValue 11157
      ProcessValue <- "Valori Temporare_Nivel Miere in Kg"
   TextField "Text field_4" at 417,16 size 147x23; Text 'Nivel Miere(Kg)'
   Switch "Switch_1" at 582,58 size 120x51; CaptionText 'Usa jos inchisa'; TextOff 'OFF'; TextOn 'ON'
      ProcessValue <- "Usi Inchise_DB_Usa jos"
   Circle "Circle_1" at 716,73 size 36x36
      Appearance <- "Usi Inchise_DB_Usa jos"
   Switch "Switch_2" at 582,136 size 120x48; CaptionText 'Usa sus inchisa'; TextOff 'OFF'; TextOn 'ON'
      ProcessValue <- "Usi Inchise_DB_Usa sus"
   Circle "Circle_2" at 715,147 size 37x37
      Appearance <- "Usi Inchise_DB_Usa sus"
   Button "Button_1" at 63,104 size 210x32; TextOff 'Setare Temperatura'
      on Press: SetBit("Valori Temporare_Setare Temperatura Manual")
      ObjectEnable <- "Valori Temporare_Mod Automat"
   TextField "Text field_5" at 159,147 size 56x23; Text 'Mixer'
   IOField "I/O field_3" at 63,184 size 96x32; FormatPattern s99999
      ProcessValue <- "Valori Temporare_Frecventa Mixer"
   TextField "Text field_6" at 164,191 size 28x23; Text 'Hz'
   Button "Button_2" at 63,231 size 211x32; TextOff 'Pornire Mixer'
      on Press: SetBit("Valori Temporare_Pornire Mixer Manual")
   TextField "Text field_7" at 130,275 size 118x23; Text 'Timp Mixare'
   IOField "I/O field_4" at 63,313 size 96x32; FormatPattern s99999
      ProcessValue <- "Valori Temporare_Setare Temporizator"
   TextField "Text field_8" at 14,316 size 42x23; Text 'Set:'
   TextField "Text field_9" at 168,316 size 80x23; Text 'Secunde'
   IOField "I/O field_5" at 260,316 size 96x32; FormatPattern s99999
      ProcessValue <- "Valori Temporare_Counter Temporizator Invers"
   TextField "Text field_10" at 15,383 size 367x23; Text 'Finalizare Program Omogenizare Miere:'
   Circle "Circle_3" at 351,382 size 34x34
      Appearance <- "Valori Temporare_Finalizare Program"
   Button "Button_3" at 63,422 size 96x32; TextOff 'Alarme'
      on Release: ActivateScreen("Alarme", 0)
   Button "Button_4" at 171,422 size 198x32; TextOff 'Grafic Temperatura'
      on Release: ActivateScreen("Istoric Temperatura", 0)
   Switch "Switch_3" at 620,406 size 120x53; CaptionText 'Start/Stop'; TextOff 'OFF'; TextOn 'ON'
      ProcessValue <- "Valori Temporare_Start/Stop"
   Circle "Circle_4" at 747,422 size 37x37
      Appearance <- "Valori Temporare_Start/Stop"
   Switch "Switch_4" at 426,403 size 120x54; CaptionText 'Switch'; TextOff 'OFF'; TextOn 'ON'
      ProcessValue <- "Valori Temporare_Mod Automat"
   Circle "Circle_5" at 548,422 size 35x35
      Appearance <- "Valori Temporare_Mod Automat"

screen "Alarme" 800x480
   AlarmView "Alarm view_1" at 24,17 size 746x327
   Button "Button_1" at 28,384 size 96x32; TextOff 'Meniu'
      on Release: ActivateScreen("Meniu", 0)
   Button "Button_2" at 136,384 size 121x32; TextOff 'Avarie Mixer'
      on Release: function_b3f726e6("Valori Temporare_Alarma Mixer", 0)
   Button "Button_3" at 135,428 size 121x32; TextOff 'Repara Mixer'
      on Release: function_a9b64e44("Valori Temporare_Alarma Mixer", 0)
   Button "Button_4" at 270,384 size 205x32; TextOff 'Avarie Senzor Presiune'
      on Release: function_b3f726e6("Valori Temporare_Alarma Senzor Presiune", 0)
   Button "Button_5" at 270,428 size 206x32; TextOff 'Repara Senzor Presiune'
      on Release: function_a9b64e44("Valori Temporare_Alarma Senzor Presiune", 0)
   Button "Button_6" at 491,384 size 246x32; TextOff 'Avarie Senzor Temperatura'
      on Release: function_b3f726e6("Valori Temporare_Alarma  Senzor Temperatura", 0)
   Button "Button_7" at 491,428 size 246x32; TextOff 'Repara Senzor Temperatura'
      on Release: function_a9b64e44("Valori Temporare_Alarma  Senzor Temperatura", 0)

screen "Istoric Temperatura" 800x480
   TrendView "Trend view_1" at 27,29 size 741x354
   Button "Button_1" at 338,410 size 96x32; TextOff 'Meniu'
      on Release: ActivateScreen("Meniu", 0)
*)